// TIA Portal V17 export
// export: Created 2025-03-10T13:12:54.0907285Z, ExportSetting WithDefaults, DisplayName Totally Integrated Automation Portal, DisplayVersion V17 Update 8, DisplayName TIA Portal Openness, DisplayVersion V17 Update 8, DisplayName TIA Portal Version Control Interface, DisplayVersion V17, DisplayName SINAMICS Startdrive Advanced, DisplayVersion V17 SP2, DisplayName SINAMICS Startdrive G110M, G120, G120C, G120D, G120P, G115D, DisplayVersion V17 SP2, DisplayName SINAMICS Startdrive G130, G150, S120, S150, SINAMICS MV, S210, DisplayVersion V17 SP2, DisplayName STEP 7 Professional, DisplayVersion V17 Update 8, DisplayName SINUMERIK ONE STEP 7 Toolbox, DisplayVersion V17 Update 12, DisplayName SINUMERIK 840D sl STEP 7 Toolbox, DisplayVersion V17 Update 12, DisplayName STEP 7 Safety, DisplayVersion V17 Update 6, DisplayName WinCC Advanced, DisplayVersion V17 Update 8
DATA_BLOCK "DB21003_POWDER_FEEDER_HMI_INTERLOCK"   // DB21003
{ S7_Optimized_Access := 'FALSE'; DB_Accessible_From_OPC_UA := 'FALSE' }
VERSION : 0.1
// stored: AutoNumber false, DBAccessibleFromOPCUA false, DBAccessibleFromWebserver true, IsOnlyStoredInLoadMemory false, IsWriteProtectedInAS false
   VAR
      POWDER_FEEDER_1_UNIT_01 : Struct
         "HMI_Values Setpoints" : "POWDER FEEDER HMI VALUES SETPOINTS";
         "HMI_Offsets Alarms and Warnings" : "POWDER FEEDER HMI OFFSETS ALARMS WARNINGS";
         HMI_ACTIONS_STATUS { S7_SetPoint := 'True'} : "POWDER FEEDER HMI ACTIONS";
      END_STRUCT;
      POWDER_FEEDER_1_UNIT_02 : Struct
         "HMI_Values Setpoints" : "POWDER FEEDER HMI VALUES SETPOINTS";
         "HMI_Offsets Alarms and Warnings" : "POWDER FEEDER HMI OFFSETS ALARMS WARNINGS";
         HMI_ACTIONS_STATUS : "POWDER FEEDER HMI ACTIONS";
      END_STRUCT;
      POWDER_FEEDER_2_UNIT_02 : Struct
         "HMI_Values Setpoints" : "POWDER FEEDER HMI VALUES SETPOINTS";
         "HMI_Offsets Alarms and Warnings" : "POWDER FEEDER HMI OFFSETS ALARMS WARNINGS";
         HMI_ACTIONS_STATUS : "POWDER FEEDER HMI ACTIONS";
      END_STRUCT;
   END_VAR
BEGIN
END_DATA_BLOCK
